PROGRAM PRG_COM_VLS
VAR
END_VAR

fbSerialLineControl(
	Mode:= SERIALLINEMODE_EL6_22B,
	pComIn:= ADR(stComIn),
	pComOut:=ADR(stComOut),
	SizeComIn:= SIZEOF(stComIn),
	TxBuffer:= SerialTXBuffer,
	RxBuffer:= SerialRXBuffer,
	Error=> ,
	ErrorID=> );

END_PROGRAM

(* stored: Version 1.1.0.1, ProductVersion 3.1.4022.18
   POU PRG_COM_VLS: Id {7c20adc9-8454-4d3d-b760-2b63ca76f659}, SpecialFunc None *)
